FUNCTION_BLOCK FB_PositionStateManager_Test EXTENDS TcUnit.FB_TestSuite
VAR
    Expected: BOOL;
    Actual: BOOL;
END_VAR

TEST('FB_PositionStateManager_Test Dummy Test');
AssertEquals(Expected := Expected,
             Actual := Actual,
             Message := 'Error Message');
TEST_FINISHED();

END_FUNCTION_BLOCK

(* stored: Version 1.1.0.1, ProductVersion 3.1.4022.18
   POU FB_PositionStateManager_Test: Id {4b536082-bb7d-4f06-8efc-8b3f61370fca}, SpecialFunc None *)
